Yaskawa INFORM job: TEST20231218.JBI

/JOB
//NAME TEST20231218
//POS
///NPOS 11,0,0,0,0,0
///TOOL 5
///POSTYPE PULSE
///PULSE
C00000=-1,-50477,-58433,3,-74929,486
C00001=-21533,8384,-65430,-73054,-31337,42440
C00002=-21533,13564,-68096,-82219,-30340,47473
C00003=-17484,12524,-69475,-84659,-28883,47530
C00004=-17485,12524,-69475,-84659,-28882,47529
C00005=-22343,25867,-50470,-59695,-46712,48966
C00006=-21029,40125,-27373,-41567,-63253,52558
C00007=-17582,47556,-14424,-31287,-72915,56096
C00008=-18208,43678,-21255,-31284,-71580,56692
C00009=-18208,40400,-19150,-30722,-74908,55693
C00010=-2,-50477,-58433,4,-74930,485
//INST
///DATE 2024/03/06 14:13
///ATTR SC,RW
///GROUP1 RB1
NOP
MOVJ C00000 VJ=5.00
MOVJ C00001 VJ=5.00
MOVJ C00002 VJ=2.00
ARCON AC=40 AVP=50
MOVL C00003 V=2.0
ARCOF
MOVC C00004 V=2.0
MOVC C00005 V=3.0
MOVC C00006 V=3.0
MOVL C00007 V=3.0
ARCON AC=40 AVP=50
MOVL C00008 V=2.0
ARCOF
MOVJ C00009 VJ=2.00
MOVJ C00010 VJ=5.00
END
